FUNCTION_BLOCK FB_SkillHandler EXTENDS FB_SKILL
VAR_INPUT
	_owner: POINTER TO FB_ROB;
END_VAR
VAR_OUTPUT
END_VAR
VAR
	activSkill: POINTER TO FB_SKILL;
	_finished: BOOL;
END_VAR

// IF activSkill^.bDone THEN
// 	_finished:=True;
// END_IF

{attribute 'TcRpcEnable':='1'}
METHOD AbortActifSkill : BOOL
VAR_INPUT
END_VAR
activSkill^.Stop();
END_METHOD

PROPERTY ActiveSkillFinished : BOOL
GET
ActiveSkillFinished := _finished;
END_GET
END_PROPERTY

{attribute 'TcRpcEnable':='1'}
METHOD CallSkill
VAR_INPUT
	pSkill : POINTER TO FB_SKILL;
	name: STRING := '';
END_VAR

VAR
	toolready: BOOL;
	i: INT;
END_VAR
IF name<>'' THEN
	FOR i := TO_INT(LOWER_BOUND(_owner^.pA_Skills, 1)) TO TO_INT(UPPER_BOUND(_owner^.pA_Skills, 1)) DO
		IF _owner^.pA_Skills[i]<>0 THEN
			IF FIND(STR1:=_owner^.pA_Skills[i]^.Name, STR2:=name)<>0 THEN
				pSkill:=_owner^.pA_Skills[i];
				ADSLOGSTR(
					msgCtrlMask := ADSLOG_MSGTYPE_HINT,
					msgFmtStr   := 'CallSkill: Found by name: %s',
					strArg      := _owner^.pA_Skills[i]^.Name
				);
				EXIT;
			END_IF
		END_IF
	END_FOR
	
END_IF


IF pSkill<>0 THEN
	activSkill:= pSkill;
	
// 	toolready:=TRUE;
// 	IF _owner^.pTool<>0 THEN
// 		toolready:=FALSE;
// 		IF _owner^.pTool^.State = eState.Active THEN
// 			toolready:=TRUE;
// 		END_IF
// 	END_IF
	
	
	pSkill^.Start();
ELSE
	ADSLOGSTR(
    msgCtrlMask := ADSLOG_MSGTYPE_ERROR,
    msgFmtStr   := 'CallSkill: Pointer to Skill is empty: %s',
    strArg      := _owner^.Path
);
END_IF
END_METHOD

PROPERTY GetActivSkill : POINTER TO FB_SKILL
GET
GetActivSkill := activSkill;
END_GET
END_PROPERTY

END_FUNCTION_BLOCK

(* stored: Version 1.1.0.1, ProductVersion 3.1.4026.18
   POU FB_SkillHandler: Id {d564b0b9-96bf-4626-9d61-904bd7d86173}, SpecialFunc None
   Method AbortActifSkill: Id {10338084-d473-478a-aa27-fc35b9873599}
   Property ActiveSkillFinished: Id {e768b71e-2b8c-4823-b6e5-97c90ef183b8}
   Get Get: Id {8bd5e583-c1a7-40cf-800c-cc46c8f2112d}
   Method CallSkill: Id {d8fc5668-9fa7-43c2-a944-aada2bd4cb8c}
   Property GetActivSkill: Id {a76ffee6-6586-41ec-827c-b1a5d3fc1e96}
   Get Get: Id {d373d262-644a-4298-ae86-7673cc4dcfd7} *)
